// TIA Portal V17 export
// export: Created 2025-03-05T08:00:04.5463532Z, ExportSetting WithDefaults, DisplayName Totally Integrated Automation Portal, DisplayVersion V17 Update 8, DisplayName TIA Portal Openness, DisplayVersion V17 Update 8, DisplayName TIA Portal Version Control Interface, DisplayVersion V17, DisplayName SINAMICS Startdrive Advanced, DisplayVersion V17 SP2, DisplayName SINAMICS Startdrive G110M, G120, G120C, G120D, G120P, G115D, DisplayVersion V17 SP2, DisplayName SINAMICS Startdrive G130, G150, S120, S150, SINAMICS MV, S210, DisplayVersion V17 SP2, DisplayName STEP 7 Professional, DisplayVersion V17 Update 8, DisplayName SINUMERIK ONE STEP 7 Toolbox, DisplayVersion V17 Update 12, DisplayName SINUMERIK 840D sl STEP 7 Toolbox, DisplayVersion V17 Update 12, DisplayName STEP 7 Safety, DisplayVersion V17 Update 6, DisplayName WinCC Advanced, DisplayVersion V17 Update 8
FUNCTION "FC2031_MACHINE_CONTINUOUS_CYCLE" : Void   // FC2031, LAD
{ S7_Optimized_Access := 'FALSE' }
AUTHOR : ETXETAR
VERSION : 1.0
// stored: AutoNumber false, IsIECCheckEnabled false, SetENOAutomatically false, UDAEnableTagReadback false
BEGIN

REGION Network 1: CONTINUOUS CYCLE SELECTED / CONTINUOS MODE
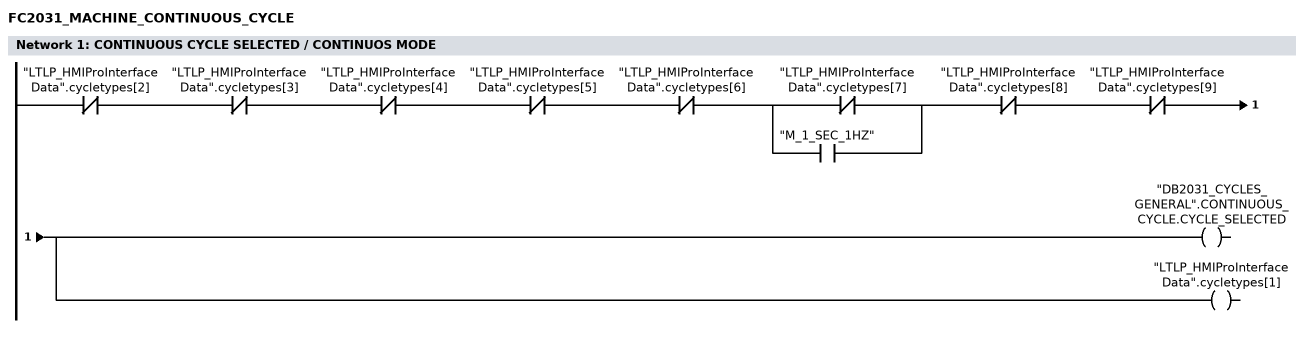
   RUNG wire#powerrail
      I_Contact( "LTLP_HMIProInterfaceData".cycletypes[2] )
      I_Contact( "LTLP_HMIProInterfaceData".cycletypes[3] )
      I_Contact( "LTLP_HMIProInterfaceData".cycletypes[4] )
      I_Contact( "LTLP_HMIProInterfaceData".cycletypes[5] )
      I_Contact( "LTLP_HMIProInterfaceData".cycletypes[6] )
      wire#w1
      I_Contact( "LTLP_HMIProInterfaceData".cycletypes[7] )
      wire#w2
      I_Contact( "LTLP_HMIProInterfaceData".cycletypes[8] )
      I_Contact( "LTLP_HMIProInterfaceData".cycletypes[9] )
      wire#w3
      Coil( "DB2031_CYCLES_GENERAL".CONTINUOUS_CYCLE.CYCLE_SELECTED )
   END_RUNG
   RUNG wire#w1
      Contact( "M_1_SEC_1HZ" )
   END_RUNG wire#w2
   RUNG wire#w3
      Coil( "LTLP_HMIProInterfaceData".cycletypes[1] )
   END_RUNG
   // the same network as SCL:
   "DB2031_CYCLES_GENERAL".CONTINUOUS_CYCLE.CYCLE_SELECTED := NOT "LTLP_HMIProInterfaceData".cycletypes[2] AND NOT "LTLP_HMIProInterfaceData".cycletypes[3] AND NOT "LTLP_HMIProInterfaceData".cycletypes[4] AND NOT "LTLP_HMIProInterfaceData".cycletypes[5] AND NOT "LTLP_HMIProInterfaceData".cycletypes[6] AND (NOT "LTLP_HMIProInterfaceData".cycletypes[7] OR "M_1_SEC_1HZ") AND NOT "LTLP_HMIProInterfaceData".cycletypes[8] AND NOT "LTLP_HMIProInterfaceData".cycletypes[9];
   "LTLP_HMIProInterfaceData".cycletypes[1] := "DB2031_CYCLES_GENERAL".CONTINUOUS_CYCLE.CYCLE_SELECTED;
END_REGION
END_FUNCTION
